// TIA Portal V16 export
// export: Created 2021-08-26T13:23:50.3138984Z, ExportSetting WithDefaults, DisplayName Totally Integrated Automation Portal, DisplayVersion V16 Update 4, DisplayName TIA Portal Version Control Interface, DisplayVersion V16 Update 2, DisplayName TIA Portal Openness, DisplayVersion V16 Update 4, DisplayName STEP 7 Professional, DisplayVersion V16 Update 4, DisplayName STEP 7 Safety, DisplayVersion V16, DisplayName WinCC Advanced, DisplayVersion V16 Update 4
FUNCTION "funkcja1" : Void   // FC1, LAD
TITLE = taki oto jest tytuł bloku
{ S7_Optimized_Access := 'TRUE' }
VERSION : 0.1
// komentarz bloku
// stored: AutoNumber false, IsIECCheckEnabled false, SetENOAutomatically false, UDAEnableTagReadback false
BEGIN

REGION Network 1: komentarz linia 1
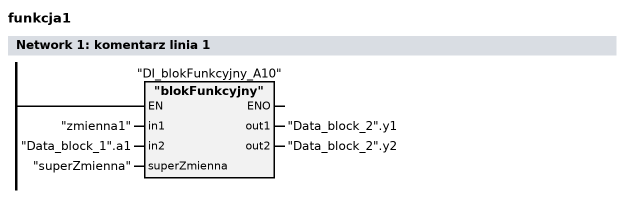
   RUNG wire#powerrail
      "DI_blokFunkcyjny_A10"(in1 := "zmienna1", in2 := "Data_block_1".a1, superZmienna := "superZmienna", out1 => "Data_block_2".y1, out2 => "Data_block_2".y2)
   END_RUNG
   // the same network as SCL:
   "DI_blokFunkcyjny_A10"(in1 := "zmienna1",   // "blokFunkcyjny"
                          in2 := "Data_block_1".a1,
                          superZmienna := "superZmienna",
                          out1 => "Data_block_2".y1,
                          out2 => "Data_block_2".y2);
END_REGION
END_FUNCTION
